// TIA Portal V18 export
FUNCTION "AHUSPCtrl" : Void   // FC60003, LAD
{ S7_Optimized_Access := 'TRUE' }
VERSION : 0.1
// stored: AutoNumber false, IsIECCheckEnabled false, SetENOAutomatically false, UDAEnableTagReadback false
   VAR_INPUT
      iUnitID : Int;
      rProtTempHeating : Real;
      rEconTempHeating : Real;
      rPreComfTempHeating : Real;
      rComfTempHeating : Real;
      rComfTempCooling : Real;
      rPreComfTempCooling : Real;
      rEconTempCooling : Real;
      rProtTempCooling : Real;
      rProtIAQ : Real;
      rEconIAQ : Real;
      rPreComfIAQ : Real;
      rComfIAQ : Real;
      rProtdP : Real;
      rEcondP : Real;
      rPreComfdP : Real;
      rComfdP : Real;
   END_VAR
   VAR_OUTPUT
      rActualTempHeating : Real;
      rActualTempCooling : Real;
      rActualIAQ : Real;
      rActualdP : Real;
   END_VAR
   VAR_TEMP
      iTargetUnitMode_old : Int;
      xResetActualOperationMode : Bool;
      iActualUnitMode_old : Int;
      xResetTargetSetpoints : Bool;
   END_VAR
BEGIN

REGION Network 1 (SCL)
   // Redefine Target Setpoints
   IF "AHUOpModes".OpModes.cActual[#iUnitID] = "AHUOpModes".OpModes.cTarget[#iUnitID] THEN // !!!Змінити на PrevOpMode
       // Statement section IF
       CASE "AHUOpModes".OpModes.cActual[#iUnitID] OF
           0:  // Protection
               "AHUSetPoints".SetPoints.Room.Target.RATHeating[#iUnitID] := #rProtTempHeating;
               "AHUSetPoints".SetPoints.Room.Target.RATCooling[#iUnitID] := #rProtTempCooling;
               "AHUSetPoints".SetPoints.Room.Target.IAQ[#iUnitID] := #rProtIAQ;
               "AHUSetPoints".SetPoints.Room.Target.BuildingdP[#iUnitID] := #rProtdP;
           1:  // Economy
               "AHUSetPoints".SetPoints.Room.Target.RATHeating[#iUnitID] := #rEconTempHeating;
               "AHUSetPoints".SetPoints.Room.Target.RATCooling[#iUnitID] := #rEconTempCooling;
               "AHUSetPoints".SetPoints.Room.Target.IAQ[#iUnitID] := #rEconIAQ;
               "AHUSetPoints".SetPoints.Room.Target.BuildingdP[#iUnitID] := #rEcondP;
           2: // Precomfort
               "AHUSetPoints".SetPoints.Room.Target.RATHeating[#iUnitID] := #rPreComfTempHeating;
               "AHUSetPoints".SetPoints.Room.Target.RATCooling[#iUnitID] := #rPreComfTempCooling;
               "AHUSetPoints".SetPoints.Room.Target.IAQ[#iUnitID] := #rPreComfIAQ;
               "AHUSetPoints".SetPoints.Room.Target.BuildingdP[#iUnitID] := #rPreComfdP;
           ELSE  // Statement section ELSE
               "AHUSetPoints".SetPoints.Room.Target.RATHeating[#iUnitID] := #rComfTempHeating;
               "AHUSetPoints".SetPoints.Room.Target.RATCooling[#iUnitID] := #rComfTempCooling;
               "AHUSetPoints".SetPoints.Room.Target.IAQ[#iUnitID] := #rComfIAQ;
               "AHUSetPoints".SetPoints.Room.Target.BuildingdP[#iUnitID] := #rComfdP;
       END_CASE;
       ;
   END_IF;
END_REGION

REGION Network 2 (SCL): Smoothing Actual Setpoints
   IF 1 THEN
       #rActualTempHeating := "AHUSetPoints".SetPoints.Room.Target.RATHeating[#iUnitID];
       #rActualTempCooling := "AHUSetPoints".SetPoints.Room.Target.RATCooling[#iUnitID];
       #rActualIAQ := "AHUSetPoints".SetPoints.Room.Target.IAQ[#iUnitID];
       #rActualdP := "AHUSetPoints".SetPoints.Room.Target.BuildingdP[#iUnitID];
   END_IF;
END_REGION
END_FUNCTION
